(* IEC 61131-3 sources: lacyccom-procedural/src/drive_functions/blocks (part 4) *)

(* ---- LAcycCom_ReadDriveMessagesOperatingHours.st ---- *)
USING System.Timer;
USING System.DateTime;
USING System.Math;
USING Siemens.Simatic.Hardware.Utilities;
USING Siemens.Simatic.Clocks;

NAMESPACE Simatic.Ax.LAcycCom.Procedural
  TYPE
    LAcycCom_ReadDriveMessagesOperatingHoursStates : SINT (
      FB_IDLE := SINT#0,   // Idle state in FB
      FB_ALARMS_DATASET := SINT#1,   // Preparing dataset state in FB (alarms)
      FB_FAULTS_DATASET := SINT#2,   // Preparing dataset state in FB (faults)
      FB_ALARMS_GONE_DATASET := SINT#4,   // State that prepare dataset (r2125) and call ReadDriveParams
      FB_READ_STEP_1 := SINT#5,   // Call ReadDriveParams and write messages in statBuffer state
      FB_READ_STEP_2 := SINT#6,   // Call ReadDriveParams with FALSE state
      FB_SORTING := SINT#10   // Sorting state in FB
    ) := FB_IDLE;
  END_TYPE

  ///------------------------------------------------------------------------------
  /// SIEMENS AG
	/// (c)Copyright 2026 All Rights Reserved
	///-----------------------------------------------------------------------------
	/// Library: LAcycCom
	/// Tested with: S7-1513-1 PN
	/// Engineering: SIMATIC AX
	/// Restrictions: The drive must provide operating hours (days + ms)
	/// Requirements: S7-1200 / S7-1500
	///               FB LAcycCom_ResourceManager is required
	/// Functionality: Read alarms and faults from G120 drive (convert operating
	///                hours to "time" in reference to SIMATIC controller) and output
	///                in structure (newest elements first)
  ///------------------------------------------------------------------------------
  FUNCTION_BLOCK LAcycCom_ReadDriveMessagesOperatingHours
    {S7.Extern = ReadWrite}
    VAR_INPUT
      execute : BOOL;   /// TRUE: Rising edge starts the functionality once
      alarms : BOOL := TRUE;   /// TRUE: Enable reading of alarms
      faults : BOOL := TRUE;   /// TRUE: Enable reading of faults
      hardwareId : UINT;   /// Hardware identifier of the hardware module
    END_VAR

    {S7.Extern = ReadOnly}
    VAR_OUTPUT
      done : BOOL;   /// TRUE: Commanded action has been completed successfully
      busy : BOOL;   /// TRUE: FB is not finished and new output values can be expected
      error : BOOL;   /// TRUE: Rising edge informs that an error occurred during the execution of the FB
      status : LAcycCom_DriveFunctionStatus;   /// Status identifier
      diagnostics : LAcycCom_typeDriveDiagnostics;   /// Diagnostics structure
      messages : ARRAY[0..MESSAGES_COUNT_UPPER_LIM] OF LAcycCom_typeDriveMessage;   /// List of drive messages
    END_VAR

    VAR_IN_OUT
      requestBufferHeader : LAcycCom_typeRequestBufferHeader;   /// Interface for header of request buffer
      requestBuffer : ARRAY[*] OF LAcycCom_typeRequestBufferElement;   /// Interface for request buffer
    END_VAR

    VAR
      _busy : BOOL;   /// Static value for output busy
      _done : BOOL;   /// Static value for output done
      _error : BOOL;   /// Static value for output error
      _status : LAcycCom_DriveFunctionStatus;   /// Static value for output status
      _executeOld : BOOL;   /// Old value of execute for edge detection
      _fbstate : LAcycCom_ReadDriveMessagesOperatingHoursStates;   /// States in the function block state machine
      _alarmsInput : BOOL;   /// Static variable for input "alarms"
      _faultsInput : BOOL;   /// Static variable for input "faults"
      _driveObjectId : SINT;   /// Intern identification number of the drive object
      _hardwareId : UINT;   /// Intern hardware identifier of the hardware module
      _dtl : LDATE_AND_TIME;   /// Time varible for comparasion (sorting)
      _indexNew : DINT;   /// Index of newest elemet (for sorting)
      _offset : SINT;   /// Offset for statBuffer/ first empty element in statBuffer
      _warningNoMessages : BOOL;   /// TRUE: At least one of two inputs must be selected
      _warningRetriggering : BOOL;   /// TRUE: Input execute is set during processing
      _alarmsComplete : BOOL;   /// TRUE: FB_READ state complete successfully (alarms)
      _currentMessage : LAcycCom_DriveMessageType;   /// Static variable represents current message type
      _cpuTime : LDATE_AND_TIME;   /// Current data and current time-of-day of the CPU clock
      _cuTimeNotRead : BOOL;   /// TRUE: r2124 (represents system runtime total of CU ) is not yet read and evaluate
      _cpuTimeNotRead : BOOL;   /// TRUE: CPU time is not yet read
      _driveObjectTOD : TIME_OF_DAY;   /// Static variable represents r2124[0] - ms, convert to TOD
      _driveObjectDays : DINT;   /// Static variable represents r2124[1] - days
      _diffDays : DINT;   /// Difference in days between actual time from system runtime counter and time from come message
      _goneAlarms : ARRAY[0..ELEMENTS_COUNT_UPPER_LIM] OF BOOL;   /// TRUE: this alarm is already gone
      _dataset : ARRAY[0..PARAMETER_COUNT_READ_UPPER_LIM] OF LAcycCom_typeDriveDataset;   /// Dataset for LAcycCom_ReadDriveParams
      _buffer : ARRAY[0..MESSAGES_COUNT_UPPER_LIM] OF LAcycCom_typeDriveMessage;   /// Buffer for store alarms, faults and SI messages
      _instReadDriveParams : LAcycCom_ReadDriveParams;   /// Instance of LAcycCom_ReadDriveParams
    END_VAR

    VAR_TEMP
      tempIndex : DINT;   // Temporary loop index variable
      tempSort : SINT;   // Temporary loop variable for sorting
      tempUInt : UINT;   // Temporary UInt variable
      tempDriveObjectDays : DINT;   // Temporary variable for days
      tempDriveObjectTOD : TIME_OF_DAY;   // Temporary variable for data type TOD
      tempDays : DINT;
      tempTOD : TIME_OF_DAY;
      tempRetValWord : WORD;   // Return value of system function
      tempQuitient : DINT;   // Temporary variable for quititent
      tempRemainder : DINT;   // Temporary variable for remainder
      tempDTL : LDATE_AND_TIME;   // Temporary DTL variable
      tempGeoAddr : GeoAddr;   // Current Geo Address information
      tempVoidDiagnostics : LAcycCom_typeDriveDiagnostics;   // Temporary empty diagnostics structure
      tempVoidMessage : LAcycCom_typeDriveMessage; // Temporary empty message structure
    END_VAR

    VAR CONSTANT
      INT_ERR_NOT_CONFIG : WORD := WORD#16#8093;   // The DP component addressed via ID or F_ID is not configured (ReadRecord/WriteRecord)
      INT_ERR_NOT_KNOWN : WORD := WORD#16#80B0;   // Data record not known in module. Illegal data record number ≥ 256 (ReadRecord/WriteRecord)
      INT_ERR_LOG_START_ADDR : WORD := WORD#16#8090;   // Invalid logical start address (ReadRecord/WriteRecord)
      DO_NOT_EXIST : WORD := WORD#16#0019;   // Drive object does not exist
      OFFSET_INFO : SINT := SINT#8;   // Offset in dataset for "info" information
      OFFSET_DAYS : SINT := SINT#16;   // Offset in dataset for "Count days" information
      OFFSET_MS : SINT := SINT#24;   // Offset in dataset for "Count ms" information
      PARAMETER_COUNT_READ_UPPER_LIM : INT := INT#33;   // Count of parameters to be read in ReadDriveParams
      ELEMENTS_COUNT_UPPER_LIM : INT := INT#7;   // Count of elements in one message type
      INIT_DATASET : BYTE := BYTE#16#FF;   // Init value for dataset.errorValue
      MAX_COUNT_DAYS : DINT := DINT#24;   // Max count of days of data type "Time"
      DRIVE_OBJECT_ID_G120 : SINT := SINT#1;   // Drive object ID for G120 (e.g. CU240)
      MESSAGES_UPPER_LIM_LOCAL : INT := INT#15;   // Upper limit of elements in LAcycCom_typeDriveMessages
      DAYS_TO_MS : DINT := DINT#86400000;   // Constant to conversion from days to ms (1000*60*60*24)
      MESSAGES_COUNT_UPPER_LIM : INT := INT#23;   // Maxmimum number of messages
      TO_NS : LREAL := LREAL#1.0e+9 * 3600 * 24;   // Conversion value for days to ns
    END_VAR

    // Check if FB is triggered
    IF (execute = TRUE) AND (_executeOld = FALSE) AND (_busy = TRUE) THEN
      // Input execute is set during processing
      status := LAcycCom_DriveFunctionStatus#WARN_EXECUTE_SET_DURING_PROCESSING;
      _warningRetriggering := TRUE;
      _executeOld := execute;

    ELSIF (execute = TRUE) AND (_executeOld = FALSE) THEN
      // First call
      // Functionality is busy
      _busy := TRUE;

      // Reset other outputs
      _error := FALSE;
      _done := FALSE;
      _status := LAcycCom_DriveFunctionStatus#STATUS_FIRST_CALL;
      status := _status;

      busy := _busy;
      error := _error;
      done := _done;
      _executeOld := execute;

      // Initialize
      _alarmsInput := alarms;
      _faultsInput := faults;
      _driveObjectId := DRIVE_OBJECT_ID_G120;
      _hardwareId := hardwareId;
      _offset := SINT#0;
      _indexNew := SINT#0;
      diagnostics := tempVoidDiagnostics;
      diagnostics.firstParameterError := -1; // V1.3.2
      diagnostics.errorValue := BYTE#16#FF; // V1.3.2
      _warningNoMessages := FALSE;
      _warningRetriggering := FALSE;
      _currentMessage := LAcycCom_DriveMessageType#ALARM;
      _alarmsComplete := FALSE;
      // Set a default value to first entry in dataset
      _dataset[0].errorValue := INIT_DATASET;
      // Set init time for comparison (sorting)
      _dtl := tempDTL;
      _cpuTimeNotRead := TRUE;
      _cuTimeNotRead := TRUE;

        // Clearing static and output area for alarms, faults and SI messages
        FOR tempIndex := 0 TO MESSAGES_COUNT_UPPER_LIM DO
          _buffer[tempIndex] := tempVoidMessage;
        END_FOR;
      // Write diagnostics
      diagnostics.hardwareId := _hardwareId;
      diagnostics.driveObjectId := _driveObjectId;

      // Call ReadDriveParams with FALSE
      _instReadDriveParams(execute := FALSE,
                          requestBufferHeader := requestBufferHeader,
                          requestBuffer := requestBuffer,
                          dataset := _dataset);

      // Check if device hardware address exist
      tempRetValWord := ReadSlotFromHardwareID(hardwareId := _hardwareId,
                                          geoAddr := tempGeoAddr);

      // Check if everything is okay
      IF tempRetValWord <> WORD#16#0 THEN
        _error := TRUE;
        diagnostics.subfunctionStatus := tempRetValWord;
        _status := LAcycCom_DriveFunctionStatus#ERR_HW_ID;
        RETURN;

      END_IF;

      // Alarms or faults
      IF _faultsInput = TRUE THEN
        _fbstate := LAcycCom_ReadDriveMessagesOperatingHoursStates#FB_FAULTS_DATASET;
      ELSIF _alarmsInput = TRUE THEN
        _fbstate := LAcycCom_ReadDriveMessagesOperatingHoursStates#FB_ALARMS_GONE_DATASET;
      ELSE
        // Warning. At least one of two inputs must be selected
        _status := LAcycCom_DriveFunctionStatus#STATUS_FINISHED_NO_MSG_SELECTED;
        _fbstate := LAcycCom_ReadDriveMessagesOperatingHoursStates#FB_SORTING;
        _warningNoMessages := TRUE;
      END_IF;
      RETURN;

    // Check if FB is disabled (falling edge) after job is done or FB is in error state
    ELSIF (execute = FALSE AND _busy = FALSE) AND
      (_error = TRUE OR _done = TRUE)
    THEN
      // Error outputs are reset with falling edge of enable input
      _error := FALSE;

      // Enable and busy are reset with falling edge of enable input
      _done := FALSE;
      _busy := FALSE;

      // Write outputs
      _status := LAcycCom_DriveFunctionStatus#STATUS_NO_CALL;
      status := _status;
      busy := _busy;
      done := _done;
      error := _error;
      _fbstate := LAcycCom_ReadDriveMessagesOperatingHoursStates#FB_IDLE;

      _executeOld := execute;
      RETURN;

      // FB is currently executed and not finished
    ELSIF _busy = TRUE THEN
      _executeOld := execute;

      // FB is disabled
    ELSE
      _executeOld := execute;
      RETURN;
    END_IF;

    //----------------------------------------------------------------------------------------------
    IF (_busy = TRUE) AND (_error = FALSE) THEN  // Functionality running
      CASE _fbstate OF

        LAcycCom_ReadDriveMessagesOperatingHoursStates#FB_ALARMS_DATASET:
          // Preparing dataset for ReadDriveParams
          // Alarms
          FOR tempIndex := 0 TO ELEMENTS_COUNT_UPPER_LIM DO
            tempUInt := TO_UINT(tempIndex);
            // Index 0 ..7 - r2122 - "Alarm Code"
            _dataset[tempIndex].parameterNumber := UINT#2122;
            _dataset[tempIndex].index := tempUInt;
            // Index 8 ..15 - r2124 - "Alarm Info"
            _dataset[tempIndex + OFFSET_INFO].parameterNumber := UINT#2124;
            _dataset[tempIndex + OFFSET_INFO].index := tempUInt;
            // Index 16 .. 23 - r2145 - "Alarm come time in days"
            _dataset[tempIndex + OFFSET_DAYS].parameterNumber := UINT#2145;
            _dataset[tempIndex + OFFSET_DAYS].index := tempUInt;
            // Index 24 .. 31 - r2123 - "Alarm come time in ms"
            _dataset[tempIndex + OFFSET_MS].parameterNumber := UINT#2123;
            _dataset[tempIndex + OFFSET_MS].index := tempUInt;
          END_FOR;
          // r2114 - System Runtime Total. Index 32 and 33
          _dataset[32].parameterNumber := UINT#2114;
          _dataset[32].index := UINT#0;    // ms
          _dataset[33].parameterNumber := UINT#2114;
          _dataset[33].index := UINT#1;  // Days
          _fbstate := LAcycCom_ReadDriveMessagesOperatingHoursStates#FB_READ_STEP_1;
          _currentMessage := LAcycCom_DriveMessageType#ALARM;

        LAcycCom_ReadDriveMessagesOperatingHoursStates#FB_FAULTS_DATASET:
          // Preparing dataset for ReadDriveParams
          // Faults
          FOR tempIndex := 0 TO ELEMENTS_COUNT_UPPER_LIM DO
            tempUInt := TO_UINT(tempIndex);
            // Index 0 ..7 - r945 - "Fault Code"
            _dataset[tempIndex].parameterNumber := UINT#945;
            _dataset[tempIndex].index := tempUInt;
            // Index 8 ..15 - r949 - "Fault Info"
            _dataset[tempIndex + OFFSET_INFO].parameterNumber := UINT#949;
            _dataset[tempIndex + OFFSET_INFO].index := tempUInt;
            // Index 16 .. 23 - r2130 - "Fault come time in days"
            _dataset[tempIndex + OFFSET_DAYS].parameterNumber := UINT#2130;
            _dataset[tempIndex + OFFSET_DAYS].index := tempUInt;
            // Index 24 .. 31 - r948 - "Fault come time in ms"
            _dataset[tempIndex + OFFSET_MS].parameterNumber := UINT#948;
            _dataset[tempIndex + OFFSET_MS].index := tempUInt;
            _goneAlarms[tempIndex] := FALSE;
          END_FOR;

          // r2114 - System Runtime Total. Index 32 and 33
          _dataset[32].parameterNumber := UINT#2114;
          _dataset[32].index := UINT#0;    // ms
          _dataset[33].parameterNumber := UINT#2114;
          _dataset[33].index := UINT#1;  // Days
          _fbstate := LAcycCom_ReadDriveMessagesOperatingHoursStates#FB_READ_STEP_1;
          _currentMessage := LAcycCom_DriveMessageType#FAULT;

        LAcycCom_ReadDriveMessagesOperatingHoursStates#FB_ALARMS_GONE_DATASET:
          IF NOT _instReadDriveParams.busy AND
            NOT _instReadDriveParams.done AND
            NOT _instReadDriveParams.error
          THEN
            // Prepare dataset
            FOR tempIndex := 0 TO ELEMENTS_COUNT_UPPER_LIM DO
              tempUInt := TO_UINT(tempIndex);
              // Index 0..7 - r2125 - "Alarm time removed in milliseconds"
              _dataset[tempIndex].parameterNumber := UINT#2125;
              _dataset[tempIndex].index := tempUInt;
            END_FOR;

          END_IF;

          // Call ReadDriveParams
          _instReadDriveParams(execute := TRUE,
                              parameterCount := ELEMENTS_COUNT_UPPER_LIM + 1, //8 parameter
                              driveObjectId := _driveObjectId,
                              hardwareId := _hardwareId,
                              requestBufferHeader := requestBufferHeader,
                              requestBuffer := requestBuffer,
                              dataset := _dataset);

          IF NOT _instReadDriveParams.busy THEN
            diagnostics := _instReadDriveParams.diagnostics;
            IF _instReadDriveParams.done = TRUE THEN
              // To determine what alarms are already gone
              FOR tempIndex := 0 TO ELEMENTS_COUNT_UPPER_LIM DO
                IF _dataset[tempIndex].dwordValue <> WORD#16#0 THEN
                  _goneAlarms[tempIndex] := TRUE;
                ELSE
                  _goneAlarms[tempIndex] := FALSE; // 01.05.02
                END_IF;
              END_FOR;

              // Call ReadDriveParams with FALSE
              _instReadDriveParams(execute := FALSE,
                                  requestBufferHeader := requestBufferHeader,
                                  requestBuffer := requestBuffer,
                                  dataset := _dataset);
              // Go next
              _fbstate := LAcycCom_ReadDriveMessagesOperatingHoursStates#FB_ALARMS_DATASET;

            ELSIF _instReadDriveParams.error = TRUE THEN
              _error := TRUE;
              // HwId is wrong
              IF (_instReadDriveParams.status = LAcycCom_DriveFunctionStatus#ERR_WRITERECORD OR _instReadDriveParams.status = LAcycCom_DriveFunctionStatus#ERR_READRECORD) AND
                ((_instReadDriveParams.diagnostics.subfunctionStatus = INT_ERR_NOT_CONFIG)
                OR (_instReadDriveParams.diagnostics.subfunctionStatus = INT_ERR_NOT_KNOWN)
                OR (_instReadDriveParams.diagnostics.subfunctionStatus = INT_ERR_LOG_START_ADDR))
              THEN
                _status := LAcycCom_DriveFunctionStatus#ERR_HW_ID;
                // Drive object does not exist
              ELSIF _dataset[0].errorValue = DO_NOT_EXIST THEN
                _status := LAcycCom_DriveFunctionStatus#ERR_DO_ID;
              ELSE
                _status := LAcycCom_DriveFunctionStatus#ERR_READ_DRIVE_PARAMS_ALARMS_GONE;

              END_IF;

            END_IF;
          END_IF;

        LAcycCom_ReadDriveMessagesOperatingHoursStates#FB_READ_STEP_1:
          IF _cpuTimeNotRead = TRUE THEN
            // Read CPU time
            tempRetValWord := GetLocalDateTime(_cpuTime); // Reading current date and time of cpu clock

            // Error occurred during RD_LOC_T command
            IF (tempRetValWord <> WORD#16#0) AND (tempRetValWord <> WORD#16#0001) THEN
              _error := TRUE;
              diagnostics.subfunctionStatus := tempRetValWord;
              _status := LAcycCom_DriveFunctionStatus#ERR_GET_LOCAL_DATE_TIME;
            END_IF;
            _cpuTimeNotRead := FALSE;
          END_IF;

          // Call ReadDriveParams
          _instReadDriveParams(execute := TRUE,
                              parameterCount := PARAMETER_COUNT_READ_UPPER_LIM + 1, //34 parameter = 32 parameter for messages + 2 parameter for "System Runtime Total" r2124[0] and r2124[1]
                              driveObjectId := _driveObjectId,
                              hardwareId := _hardwareId,
                              requestBufferHeader := requestBufferHeader,
                              requestBuffer := requestBuffer,
                              dataset := _dataset);

          IF NOT _instReadDriveParams.busy THEN
            diagnostics := _instReadDriveParams.diagnostics;
            IF _instReadDriveParams.done = TRUE THEN
              // CU Time from parameter r2124
              IF _cuTimeNotRead = TRUE THEN
                _driveObjectDays := TO_DINT(_dataset[33].dwordValue);   // Days as DINT
                _driveObjectTOD := TO_TOD(TO_LWORD(TO_LINT(_dataset[32].dwordValue) * LINT#1000000)); // ms convert to TOD
                _cuTimeNotRead := FALSE;
              END_IF;
              // Copy to static area only elements with content
              FOR tempIndex := 0 TO ELEMENTS_COUNT_UPPER_LIM DO
                IF NOT _goneAlarms[tempIndex] THEN
                  _buffer[_offset].code := TO_UINT(_dataset[tempIndex].dwordValue);
                  // If parameter empty - then go next
                  IF _dataset[tempIndex].dwordValue = WORD#16#0 THEN
                    EXIT;
                  END_IF;

                  _buffer[_offset].info := TO_UDINT(_dataset[tempIndex + OFFSET_INFO].dwordValue);
                  tempDriveObjectDays := TO_DINT(_dataset[tempIndex + OFFSET_DAYS].dwordValue);
                  tempDriveObjectTOD := TO_TOD(TO_LWORD(_dataset[tempIndex + OFFSET_MS].dwordValue));
                  //=======================================================================================================================================
                  // Calcutation "come Date and Time" of G120. This CUs (all G120 except CU230P-2) have only system runtime counter...
                  // comeDateAndTime = CPU Time(statCPUTime) - (difference statCUDays and tempDays) - (difference statCUTOD and tempTOD)
                  _diffDays := _driveObjectDays - tempDriveObjectDays; // Difference in days between actual time from system runtime counter and time from come message
                  _buffer[_offset].comeDateAndTime := _cpuTime;
                  IF ABS(_diffDays) <= MAX_COUNT_DAYS THEN  // Max value of variable Time is T#24d
                    tempDays := (TO_DINT(TO_LWORD(_buffer[_offset].comeDateAndTime)) / DAYS_TO_MS) - _diffDays; // Difference drive object days to diff days
                    tempTOD := TO_TOD(_buffer[_offset].comeDateAndTime); // extract time of day from buffer
                    NewDateAndTime(TO_LDATE(TO_LWORD(tempDays)), TO_LTOD(tempTOD), _buffer[_offset].comeDateAndTime); // create new date and time based on day difference and current time of day

                  ELSE // When count of days > 24 then must be sliced
                    tempQuitient := _diffDays / MAX_COUNT_DAYS;
                    tempRemainder := _diffDays MOD MAX_COUNT_DAYS;
                    FOR tempSort := 1 TO TO_SINT(tempQuitient) DO
                      tempDays := (TO_DINT(TO_LWORD(_buffer[_offset].comeDateAndTime)) / DAYS_TO_MS) - (MAX_COUNT_DAYS * DAYS_TO_MS);
                      tempTOD := TO_TOD(_buffer[_offset].comeDateAndTime); // extract time of day from buffer
                      NewDateAndTime(TO_LDATE(TO_LWORD(tempDays)), TO_LTOD(tempTOD), _buffer[_offset].comeDateAndTime); // create new date and time based on day difference and current time of day
                    END_FOR;
                    tempDays := (TO_DINT(TO_LWORD(_buffer[_offset].comeDateAndTime)) / DAYS_TO_MS) - (tempRemainder * DAYS_TO_MS); // Difference statCUDays and tempDays in format Time
                    tempTOD := TO_TOD(_buffer[_offset].comeDateAndTime); // extract time of day from buffer
                    NewDateAndTime(TO_LDATE(TO_LWORD(tempDays)), TO_LTOD(tempTOD), _buffer[_offset].comeDateAndTime);
                  END_IF;

                  // tempTime := T_DIFF(IN1 := statDriveObjectTOD, IN2 := tempDriveObjectTOD); // Difference statCUTOD and tempTOD in format Time - ms
                  // statBuffer.comeDateAndTime[statOffset] := T_SUB(IN1 := statBuffer.comeDateAndTime[statOffset], IN2 := tempTime); // Subtraction ms

                  tempDays := TO_DINT(TO_LWORD(_driveObjectTOD)) - TO_DINT(TO_LWORD(tempDriveObjectTOD)) / DAYS_TO_MS; // Difference statCUTOD and tempTOD in format Time - ms
                  tempTOD := TO_TOD(_buffer[_offset].comeDateAndTime); // extract time of day from buffer
                  NewDateAndTime(TO_LDATE(TO_LWORD(tempDays)), TO_LTOD(tempTOD), _buffer[_offset].comeDateAndTime);

                  //=======================================================================================================================================
                  _buffer[_offset].messageType := _currentMessage; // Identifier for message
                  _offset := _offset + SINT#1;
                END_IF;
              END_FOR;
              // Set "complete" flag
              IF _currentMessage = LAcycCom_DriveMessageType#ALARM THEN
                _alarmsComplete := TRUE;
              END_IF;

              // Go next step
              _fbstate := LAcycCom_ReadDriveMessagesOperatingHoursStates#FB_READ_STEP_2;

              // Error while reading  with ReadDriveParams
            ELSIF _instReadDriveParams.error = TRUE THEN
              _error := TRUE;
              // HwId is wrong
              IF (_instReadDriveParams.status = LAcycCom_DriveFunctionStatus#ERR_WRITERECORD OR _instReadDriveParams.status = LAcycCom_DriveFunctionStatus#ERR_READRECORD) AND
                ((_instReadDriveParams.diagnostics.subfunctionStatus = INT_ERR_NOT_CONFIG)
                OR (_instReadDriveParams.diagnostics.subfunctionStatus = INT_ERR_NOT_KNOWN)
                OR (_instReadDriveParams.diagnostics.subfunctionStatus = INT_ERR_LOG_START_ADDR))
              THEN
                _status := LAcycCom_DriveFunctionStatus#ERR_HW_ID;
                // Drive object does not exist
              ELSIF _dataset[0].errorValue = DO_NOT_EXIST THEN
                _status := LAcycCom_DriveFunctionStatus#ERR_DO_ID;
              ELSE
                CASE _currentMessage OF
                  LAcycCom_DriveMessageType#ALARM:
                    _status := LAcycCom_DriveFunctionStatus#ERR_READ_DRIVE_PARAMS_ALARMS;
                  LAcycCom_DriveMessageType#FAULT:
                    _status := LAcycCom_DriveFunctionStatus#ERR_READ_DRIVE_PARAMS_FAULTS;
                  ELSE
                    ;
                END_CASE;
              END_IF;
            END_IF;
          END_IF;

          LAcycCom_ReadDriveMessagesOperatingHoursStates#FB_READ_STEP_2:
          // Call ReadDriveParams with FALSE
          _instReadDriveParams(execute := FALSE,
                              requestBufferHeader := requestBufferHeader,
                              requestBuffer := requestBuffer,
                              dataset := _dataset);

          // Choice next step. Right call order: faults, alarms
          IF (_alarmsInput AND NOT _alarmsComplete) THEN
            _fbstate := LAcycCom_ReadDriveMessagesOperatingHoursStates#FB_ALARMS_GONE_DATASET;
          ELSE
            _fbstate := LAcycCom_ReadDriveMessagesOperatingHoursStates#FB_SORTING;
          END_IF;

        LAcycCom_ReadDriveMessagesOperatingHoursStates#FB_SORTING:
          // When at least one message has been read
          IF _offset <> 0 THEN
            // Sorting algorithm. Newest message - first
            // When more then two messages of different type have the same come time, then order sequence is - alarms, faults, SI messages
            FOR tempSort := 0 TO (_offset - SINT#1) DO
              // Find newest element
              FOR tempIndex := 0 TO (_offset - 1) DO
                IF _buffer[tempIndex].comeDateAndTime >= _dtl THEN
                  _dtl := _buffer[tempIndex].comeDateAndTime;
                  _indexNew := tempIndex;
                END_IF;
              END_FOR;

              // Copy found element to output structure
              messages[tempSort] := _buffer[_indexNew];

              // Remove this element from buffer - by setting the value as small as possible
              _buffer[_indexNew].comeDateAndTime := tempDTL;
              // Set init time for next comparison
              _dtl := tempDTL;
            END_FOR;
          END_IF;
          // Set "done" flag
          _done := TRUE;

        ELSE
          _error := TRUE;
          _status := LAcycCom_DriveFunctionStatus#ERR_UNDEFINED_STATE;
      END_CASE;
    END_IF;

    //----------------------------------------------------------------------------------------------
    // Write outputs and error handling
    //----------------------------------------------------------------------------------------------
    // Error occurred in request
    IF _error = TRUE
    THEN
      _done := FALSE;
      _busy := FALSE;
      // Write diagnostics
      diagnostics.stateNumber := _fbstate;
      diagnostics.status := _status;

      // Request finished
    ELSIF _done = TRUE
    THEN
      _busy := FALSE;
      _error := FALSE;
      _fbstate := LAcycCom_ReadDriveMessagesOperatingHoursStates#FB_IDLE;
      // Set status
      IF _warningRetriggering = TRUE THEN
        // If input execute is set during processing
        _status := LAcycCom_DriveFunctionStatus#ERR_AMBIGUOUS_FB_CALL;
        diagnostics.status := _status;
        _error := TRUE;
        _done := FALSE;
      ELSIF _warningNoMessages = FALSE THEN
        // Execution finished without errors
        _status := LAcycCom_DriveFunctionStatus#STATUS_EXECUTION_FINISHED;
      ELSE
        // Warning. At least one of two inputs must be selected
        _status := LAcycCom_DriveFunctionStatus#STATUS_FINISHED_NO_MSG_SELECTED;
        diagnostics.status := _status;
      END_IF;

      // If input execute is set during processing
    ELSIF _warningRetriggering = TRUE
    THEN
      _status := LAcycCom_DriveFunctionStatus#WARN_EXECUTE_SET_DURING_PROCESSING;

      // Request in execution
    ELSE
      _status := LAcycCom_DriveFunctionStatus#STATUS_SUBSEQUENT_CALL;
    END_IF;

    // Write static values to outputs
    done := _done;
    busy := _busy;
    error := _error;
    status := _status;
  //----------------------------------------------------------------------------------------------
  END_FUNCTION_BLOCK
END_NAMESPACE

(* ---- LAcycCom_ReadDriveParams.st ---- *)
USING System.Timer;
USING Siemens.Simatic.DistributedIO;

NAMESPACE Simatic.Ax.LAcycCom.Procedural
  TYPE INTERNAL
    LAcycCom_ReadDriveParamsStates : SINT(
      FB_IDLE := SINT#0,   // Idle state in FB
      FB_FIRST_CYCLE := SINT#1,   // First cycle state in FB
      FB_ALLOCATE := SINT#2,   // Allocating a request element in request buffer DB
      FB_GET_RESOURCE := SINT#3,   // State to check if the communication to the drive object can be established
      FB_BUSY := SINT#4,   // Busy state in FB
      FB_RELEASE := SINT#5,   // State to return the allocated index
      FB_DONE := SINT#6,   // Done state in FB
      FB_ERROR := SINT#7,   // Error state in FB
      FB_BUSY_WriteRecord := SINT#8,   // WriteRecord in busy state
      FB_BUSY_ReadRecord := SINT#9,   // ReadRecord in busy state
      FB_BUSY_WAIT := SINT#10   // State when temporary error occurred
    ) := FB_IDLE;
  END_TYPE

  ///------------------------------------------------------------------------------------------
  /// SIEMENS AG
	/// (c)Copyright 2026 All Rights Reserved
	///------------------------------------------------------------------------------------------
	/// Library: LAcycCom
	/// Tested with: S7-1513-1 PN
	/// Engineering: SIMATIC AX
	/// Restrictions: ---
	/// Requirements: S7-1200 / S7-1500
	///               FB LAcycCom_ResourceManager is required
	/// Functionality: Reads parameters from a drive object according to the configured dataset
  ///------------------------------------------------------------------------------------------
  FUNCTION_BLOCK LAcycCom_ReadDriveParams
    {S7.extern = ReadWrite}
    VAR_INPUT
      execute : BOOL;   /// TRUE: Rising edge starts the functionality once
      parameterCount : INT := -1;   /// Count of parameters to read (-1: read all parameter in dataset)
      driveObjectId : INT := -1;   /// Optional: Identification number of the drive object (value <0: driveObjectId is not used, i.e. the corresponding drive object is only addressed via the hardwareId)
      hardwareId : UINT;   /// Hardware identifier of the hardware module
    END_VAR

    {S7.extern = ReadOnly}
    VAR_OUTPUT
      done : BOOL;   /// TRUE: Finished reading all parameters
      busy : BOOL;   /// TRUE: FB is not finished and new output values can be expected
      error : BOOL;   /// TRUE: Rising edge informs that an error occurred during the execution of the FB
      status : LAcycCom_DriveFunctionStatus;   /// Status identifier
      diagnostics : LAcycCom_typeDriveDiagnostics;   /// Diagnostics structure
    END_VAR

    VAR_IN_OUT
      requestBufferHeader : LAcycCom_typeRequestBufferHeader;   /// Interface for header of request buffer
      requestBuffer : ARRAY[*] OF LAcycCom_typeRequestBufferElement;   /// Interface for request buffer
      dataset : ARRAY[*] OF LAcycCom_typeDriveDataset;   /// Interface for dataset
    END_VAR

    VAR
      _executeOld : BOOL := FALSE;   /// TRUE: Indicates that the execute input in the previous cycle was set
      _busy : BOOL := FALSE;   /// Static value for output busy
      _done : BOOL := FALSE;   /// Static value for output done
      _error : BOOL := FALSE;   /// Static value for output error
      _cmdBusy : BOOL := FALSE;   /// TRUE: Process is not yet complete
      _cmdDone : BOOL := FALSE;   /// TRUE: Data record was transferred
      _cmdError : BOOL := FALSE;   /// TRUE: An error occurred during processing
      _timerStart : BOOL := FALSE;   /// TRUE: Starts OnDelay
      _hwId : UINT := UINT#0;   /// Intern hardware identifier of the hardware module
      _doId : BYTE := BYTE#16#00;   /// Intern identification number of the drive object
      _refNo : BYTE := BYTE#16#00;   /// Reference number of request
      _withoutResourceManager : BOOL := FALSE;   /// TRUE: No resource manager available; FALSE: Resource manager available
      _fbState : LAcycCom_ReadDriveParamsStates := LAcycCom_ReadDriveParamsStates#FB_IDLE;   /// States in the function block state machine
      _fbSubState : LAcycCom_ReadDriveParamsStates := LAcycCom_ReadDriveParamsStates#FB_BUSY_WriteRecord;   /// States in the function block during processing (busy state)
      _fbSubStateOld : LAcycCom_ReadDriveParamsStates := LAcycCom_ReadDriveParamsStates#FB_BUSY_WriteRecord;   /// Previous state when temporary error occurs
      _stateNumber : LAcycCom_ReadDriveParamsStates := LAcycCom_ReadDriveParamsStates#FB_IDLE;   /// State of the FB when error occurred
      _status : LAcycCom_DriveFunctionStatus := LAcycCom_DriveFunctionStatus#STATUS_NO_CALL;   /// Static value for output status
      _subfunctionStatus : WORD := WORD#16#0000;   /// Block status or error information
      _errorCount : UINT := UINT#0;   /// Error counter of retry request
      _allocatedIndex : INT := 0;   /// Allocated element index in the buffer DB
      _countOfElements : INT := 0;   /// Number of parameters in the dataset
      _firstParameterError : INT := -1;   /// Number of parameter at which the error occurred (-1: no parameter with error)
      _warningRetriggering : BOOL;   /// TRUE: Input execute is set during processing
      _dataRecordNo : DInt;   /// Used data record
      _lowerBoundDataSet : DINT;   /// Lower bound of dataset
      _upperBoundDataSet : DINT;   /// Upper bound of dataset
      _parameter : ARRAY[0..READ_PARAMETERS_UPPER_LIM] OF LAcycCom_typeParameter;
      _reqParameterInit : LAcycCom_typeParameterAddress := ( attribute := BYTE#16#10, elementNo := BYTE#16#01, parameterNo := UINT#0, index := UINT#0 );
      _reqParameterHeader : LAcycCom_typeParameterHeader;
      _reqParameterAddress : ARRAY[0..READ_PARAMETERS_UPPER_LIM] OF LAcycCom_typeParameterAddress;
      _respParameterHeader : LAcycCom_typeParameterHeader;
      _respParameterData : ARRAY[0..LENGTH_PARAMETER_TELEGRAM_UPPER_LIM] OF BYTE;
      _instWriteRecord : WriteRecord;   /// WriteRecord command
      _instReadRecord : ReadRecord;   /// ReadRecord command
      _instOnDelay : OnDelay;   /// OnDelay
    END_VAR

    VAR_TEMP
      tempExecute : BOOL;   // TRUE: Indicates that the execute input was set
      tempCmdValid : BOOL;   // TRUE: New data record was received and is valid
      tempStatusWord : WORD;   // Temporary status
      tempUDint : UDINT;   // Temporary udint variable
      tempWord : WORD;   // Temporary word variable
      tempParameterCount : INT;   // Temporary variable of the output parameterCount
      tempPointer : INT;   // Temporary pointer variable
      tempIndex : INT;   // Temporary loop index variable
      tempLastQueueElement : INT;   // Last element in queue
      tempCmdStatus : DWORD;   // Temporary status of WriteRecord and ReadRecord command
      tempDWord : DWORD;   // Temporary DWORD variable
      tempVoidDiagnostics : LAcycCom_typeDriveDiagnostics;   // Temporary empty diagnostics structure
      tempVoidHeader : LAcycCom_typeParameterHeader;   // Temporary empty header structure
      tempActualElement : LAcycCom_typeDriveDataset;   // Temporary element of the dataset
      tempRecord : ARRAY[0..239] OF BYTE;   // Temporary record buffer for WriteRecord and ReadRecord instruction
    END_VAR

    VAR CONSTANT
      NO_PARAMETER_ERROR : INT := -1;   // No parameter error in response telegram
      ALL_ELEMENTS_OCCUPIED : INT := -1;   // All buffer elements are occupied
      READ_PARAMETERS_UPPER_LIM : INT := 38;   // Maximum count of parameters
      LENGTH_PARAMETER_TELEGRAM_UPPER_LIM : INT := 233;   // Maximum length of telegram for parameter information in BYTE
      MAX_ERROR_COUNT : UINT := UINT#40;   // Maximum error counter
      TIMER_TEMP_ERROR : TIME := T#200MS;   // Waiting time until next system function block call
      TIMER_ALLOCATION : TIME := T#10S;   // Timer limit for allocating a request element
      MAX_DRIVE_OBJECT_NO : INT := 254;   // Maximum drive object number limited by SINAMICS p101
    END_VAR

    tempExecute := execute;

    //----------------------------------------------------------------------
    // Processing
    //----------------------------------------------------------------------
    // Rising edge of execute starts functionality
    IF (tempExecute = TRUE) AND (_executeOld = FALSE) AND (_busy = TRUE) THEN
      // Input execute is set during processing
      _status := LAcycCom_DriveFunctionStatus#WARN_EXECUTE_SET_DURING_PROCESSING;
      _warningRetriggering := TRUE;

    ELSIF (tempExecute = TRUE) AND (_executeOld = FALSE) THEN
      // First call
      // Initialisation
      _done := FALSE;
      _busy := TRUE;
      _error := FALSE;
      _countOfElements := 0;
      _allocatedIndex := 0;
      _hwId := UINT#0;
      _subfunctionStatus := WORD#16#0;
      _doId := BYTE#0;
      _dataRecordNo := 0;
      _stateNumber := LAcycCom_ReadDriveParamsStates#FB_IDLE;
      _firstParameterError := -1;
      _cmdBusy := FALSE;
      _cmdDone := FALSE;
      _cmdError := FALSE;
      _errorCount := UINT#0;
      _warningRetriggering := FALSE;
      _fbSubState := LAcycCom_ReadDriveParamsStates#FB_BUSY_WriteRecord;
      _fbState := LAcycCom_ReadDriveParamsStates#FB_FIRST_CYCLE;

      _instOnDelay(signal := FALSE,
             duration := TIMER_ALLOCATION);

      // Initialize boundaries of dataset
      _lowerBoundDataSet := LOWER_BOUND(dataset, 1);
      _upperBoundDataSet := UPPER_BOUND(dataset, 1);
      _countOfElements := TO_INT(GetCountOfElements(_lowerBoundDataSet, _upperBoundDataSet));

      // FB is currently inactive
    ELSIF (tempExecute = FALSE) AND (_busy = FALSE)
    THEN
      _error := FALSE;
      _busy := FALSE;
      _done := FALSE;
      _fbState := LAcycCom_ReadDriveParamsStates#FB_IDLE;

      IF ((_status = LAcycCom_DriveFunctionStatus#WARN_EXECUTE) AND (execute = FALSE)) OR (_status <> LAcycCom_DriveFunctionStatus#WARN_EXECUTE) THEN
        _status := LAcycCom_DriveFunctionStatus#STATUS_NO_CALL;
      END_IF;

    END_IF; // tempExecute AND statExecuteOld = FALSE

    //----------------------------------------------------------------------
    // State Machine
    //----------------------------------------------------------------------

    IF (_busy = TRUE) AND (_error = FALSE) THEN  // Functionality running
      CASE _fbState OF
        LAcycCom_ReadDriveParamsStates#FB_FIRST_CYCLE:  // First cycle state

          // Clearing the sending buffer
          _reqParameterHeader := tempVoidHeader;
          FOR tempIndex := 0 TO READ_PARAMETERS_UPPER_LIM DO
            _reqParameterAddress[tempIndex] := _reqParameterInit;
          END_FOR;

          // Clearing the receive buffer
         _respParameterHeader := tempVoidHeader;
          FOR tempIndex := 0 TO LENGTH_PARAMETER_TELEGRAM_UPPER_LIM DO
            _respParameterData[tempIndex] := BYTE#16#00;
          END_FOR;

          // Initialization after start
          IF driveObjectId < 0 THEN // V1.5
            _dataRecordNo := DINT#16#B02E; // Base Mode Parameter Access local; doId not relevant
            _doId := BYTE#0;

          ELSIF (driveObjectId <= MAX_DRIVE_OBJECT_NO)
            AND (driveObjectId <> 0)
          THEN // V1.5.2
            _dataRecordNo := 47; // Data record 47; Base Mode Parameter Access global
            _doId := TO_BYTE(driveObjectId);

          ELSE // V1.5.2
            // Wrong drive object ID at input
            _error := TRUE;
            _stateNumber := _fbState;
            _status := LAcycCom_DriveFunctionStatus#ERR_INVALID_DRIVE_OBJECT_ID;
            _fbState := LAcycCom_ReadDriveParamsStates#FB_ERROR;
          END_IF;

          _hwId := hardwareId;
          tempParameterCount := parameterCount;

          diagnostics := tempVoidDiagnostics;
          IF _status = LAcycCom_DriveFunctionStatus#WARN_EXECUTE THEN
            diagnostics.status := _status;
          END_IF;

          diagnostics.driveObjectId := TO_SINT(_doId);
          diagnostics.hardwareId := _hwId;
          diagnostics.firstParameterError := _firstParameterError; // V1.3.2
          diagnostics.errorValue := BYTE#16#FF; // V1.3.2

          // Reference number for next request
          _refNo := TO_BYTE(TO_UINT(_refNo) + UINT#1);

          IF _error THEN // V1.5.2: Check if error appeared
            ;

          // Next state is depending on the FB mode
          ELSIF (_withoutResourceManager = FALSE) THEN
            _status := LAcycCom_DriveFunctionStatus#STATUS_ALLOCATE;
            _fbState := LAcycCom_ReadDriveParamsStates#FB_ALLOCATE;

          ELSE
            _status := LAcycCom_DriveFunctionStatus#STATUS_BUSY;
            _fbState := LAcycCom_ReadDriveParamsStates#FB_BUSY;
            _fbSubState := LAcycCom_ReadDriveParamsStates#FB_BUSY_WriteRecord;
          END_IF;

          // Calculates the amount of parameters (only if no error occurs)
          IF (_error = FALSE) THEN
            // Calculates the count of elements in readDataset if numberOfParameters < 1
            IF (tempParameterCount < 1) AND
              (_countOfElements <= READ_PARAMETERS_UPPER_LIM)
            THEN
              diagnostics.parameterCount := _countOfElements;
            ELSIF (tempParameterCount >= 1) AND  // V1.3.2
              // Check if numberOfParameters <= 39
              (tempParameterCount <= READ_PARAMETERS_UPPER_LIM + 1) AND
              (_countOfElements >= tempParameterCount)
            THEN
              _countOfElements := tempParameterCount;
              diagnostics.parameterCount := _countOfElements;
            ELSE
              _error := TRUE;
              _stateNumber := _fbState;
              _status := LAcycCom_DriveFunctionStatus#ERR_NO_OF_PARAMETERS;
              _fbState := LAcycCom_ReadDriveParamsStates#FB_ERROR;
            END_IF;
          END_IF; // IF (statError = FALSE)

        LAcycCom_ReadDriveParamsStates#FB_ALLOCATE:
          // Allocation of a request element
          IF (requestBufferHeader.lockBuffer = FALSE) AND (requestBufferHeader.nextFreeElement >= requestBufferHeader.bufferLowerBound) AND (requestBufferHeader.nextFreeElement <= requestBufferHeader.bufferUpperBound) THEN
            requestBufferHeader.lockBuffer := TRUE;
            _allocatedIndex := requestBufferHeader.nextFreeElement;
            requestBuffer[_allocatedIndex].state := BYTE#16#00;
            requestBuffer[_allocatedIndex].state.%X0 := TRUE;
            requestBuffer[_allocatedIndex].hardwareId := _hwId;
            requestBuffer[_allocatedIndex].queueElementNext := -1;
            _timerStart := FALSE;
            _status := LAcycCom_DriveFunctionStatus#STATUS_GET_RESOURCE;
            _fbState := LAcycCom_ReadDriveParamsStates#FB_GET_RESOURCE;

            // Build up queue
            IF (requestBufferHeader.firstQueueElement >= 0) THEN
              // Find last queue element
              tempIndex := requestBufferHeader.firstQueueElement;
              WHILE (tempIndex >= 0) DO
                tempLastQueueElement := tempIndex;
                tempIndex := requestBuffer[tempIndex].queueElementNext;
              END_WHILE;

              // Insert into list after last element
              requestBuffer[tempLastQueueElement].queueElementNext := _allocatedIndex;
              requestBuffer[_allocatedIndex].queueElementPrevious := tempLastQueueElement;
            ELSE
              // Element is first element in queue
              requestBufferHeader.firstQueueElement := _allocatedIndex;
              requestBuffer[_allocatedIndex].queueElementPrevious := -1;
            END_IF;

            // Searching for the next free request element
            FOR tempIndex := requestBufferHeader.bufferLowerBound TO TO_INT(requestBufferHeader.bufferUpperBound) DO
              IF (requestBuffer[tempIndex].state.%X0 = FALSE) THEN
                requestBufferHeader.nextFreeElement := tempIndex;
                EXIT;
              END_IF;

              // All request elements are occupied
              IF (tempIndex = requestBufferHeader.bufferUpperBound) THEN
                requestBufferHeader.nextFreeElement := ALL_ELEMENTS_OCCUPIED;
              END_IF;
            END_FOR;

            requestBufferHeader.lockBuffer := FALSE;

          ELSIF (_instOnDelay.output = TRUE) THEN
            _error := TRUE;
            _stateNumber := _fbState;
            _status := LAcycCom_DriveFunctionStatus#ERR_ALLOCATION_TIME;
            _fbState := LAcycCom_ReadDriveParamsStates#FB_ERROR;

          ELSE
            ; // Waiting until lockbit is reset and a request element is available
          END_IF; // (buffer.lockBuffer = FALSE) AND (buffer.actualWriteIndex >= 0)

          _instOnDelay(signal := _timerStart,
                 duration := TIMER_ALLOCATION);

          _timerStart := TRUE;
          IF (_instOnDelay.output = TRUE) THEN
            _timerStart := FALSE;
          END_IF;

        LAcycCom_ReadDriveParamsStates#FB_GET_RESOURCE:

          // Check buffer index for correctness
          IF (_allocatedIndex < requestBufferHeader.bufferLowerBound) OR (_allocatedIndex > requestBufferheader.bufferUpperBound) THEN
            _error := TRUE;
            _stateNumber := _fbState;
            _status := LAcycCom_DriveFunctionStatus#ERR_INVALID_BUF_INDEX;
            _fbState := LAcycCom_ReadDriveParamsStates#FB_ERROR;

          ELSE
            IF (requestBuffer[_allocatedIndex].state.%X0 = FALSE) OR
              (requestBuffer[_allocatedIndex].state.%X3 = TRUE)
            THEN
              // Request was rejected by buffer manager
              _error := TRUE;
              _stateNumber := _fbState;
              _status := LAcycCom_DriveFunctionStatus#ERR_REQUEST_REJECTED;
              _fbState := LAcycCom_ReadDriveParamsStates#FB_ERROR;

            ELSIF (requestBuffer[_allocatedIndex].state.%X2 = TRUE) THEN
              // Request already released
              _error := TRUE;
              _stateNumber := _fbState;
              _status := LAcycCom_DriveFunctionStatus#ERR_RESOURCE_RELEASED;
              _fbState := LAcycCom_ReadDriveParamsStates#FB_ERROR;

            ELSIF (requestBuffer[_allocatedIndex].state.%X1 = TRUE) THEN
              // Element is enabled
              _status := LAcycCom_DriveFunctionStatus#STATUS_BUSY;
              _fbState := LAcycCom_ReadDriveParamsStates#FB_BUSY;
              _fbSubState := LAcycCom_ReadDriveParamsStates#FB_BUSY_WriteRecord;

            ELSE
              // Element not enabled yet
              //
              _status := LAcycCom_DriveFunctionStatus#STATUS_GET_RESOURCE;
            END_IF;

          END_IF;

        LAcycCom_ReadDriveParamsStates#FB_BUSY:

          IF ((requestBuffer[_allocatedIndex].state.%X1 = TRUE) AND (_withoutResourceManager = FALSE) AND
            (requestBuffer[_allocatedIndex].state.%X3 = FALSE)) OR (_withoutResourceManager = TRUE)
          THEN
            CASE _fbSubState OF
              LAcycCom_ReadDriveParamsStates#FB_BUSY_WriteRecord:  // Writing the dataset configuration into the drive object

                IF (_cmdBusy = FALSE) THEN
                  // Resets WriteRecord command
                  _instWriteRecord(request := FALSE,
                               record := tempRecord);

                  // Creating header data
                  _reqParameterHeader.refNo := _refNo; // Telegram reference number
                  _reqParameterHeader.reqId := BYTE#16#01;  // 0x01 = request parameters
                  _reqParameterHeader.doId := _doId;  // Drive object identification number
                  _reqParameterHeader.parameterNo := TO_BYTE(_countOfElements);  // Count of parameters

                  // Copying the dataset into a static variable
                  FOR tempIndex := 0 TO _countOfElements - 1 DO
                    // begin at lower bound of dataset
                    tempActualElement := dataset[tempIndex + _lowerBoundDataSet];

                    // write common parameters
                    _parameter[tempIndex].index := tempActualElement.index;
                    _parameter[tempIndex].parameterNo := tempActualElement.parameterNumber;
                    _reqParameterAddress[tempIndex].index := _parameter[tempIndex].index;  // Subindex of parameter
                    _reqParameterAddress[tempIndex].parameterNo := _parameter[tempIndex].parameterNo;  // Parameter number
                  END_FOR;
                END_IF; // statCmdBusy = FALSE

                SerializeParamAddress(header := _reqParameterHeader, address := _reqParameterAddress, buffer := tempRecord);

                // WriteRecord command
                _instWriteRecord(request := TRUE,             // Transfer data record
                             hardwareId := _hwId,      // ID number of the hardware component
                             index := _dataRecordNo,   // Data record number
                             length := UINT#0,            // Maximum length of the data record to be transferred in bytes
                             record := tempRecord,        // Data record
                             done => _cmdDone,         // Data record was transferred
                             busy => _cmdBusy,         // The writing process is not yet complete
                             error => _cmdError,       // An error occurred during the writing process
                             status => tempCmdStatus);    // Status[1] = Error => Status[2] Error Decode + Status[3] Error Code

                // Error occurred
                IF (_cmdError = TRUE) AND (_error = FALSE) THEN
                  tempStatusWord.%B0 := tempCmdStatus.%B1;
                  tempStatusWord.%B1 := tempCmdStatus.%B2;

                  //Temporary command status (80A1, 80A7, 80B5, 80C0, 80C1, 80C2, 80C3 oder 80C4) are valid and retry command
                  IF (tempStatusWord = WORD#16#80A1) OR  // Negative acknowledgment when writing to the module
                    (tempStatusWord = WORD#16#80A7) OR   // DP slave or module is occupied (temporary error)
                    (tempStatusWord = WORD#16#80B5) OR   // DP slave or module not ready
                    (tempStatusWord = WORD#16#80C0) OR   // The data can only be written when the CPU is in STOP mode. Note: this means that writing by the user program is not possible. You can only write the data online with PG/PC.
                    (tempStatusWord = WORD#16#80C1) OR   // The data of the previous write job on the module for the same data record have not yet been processed by the module.
                    (tempStatusWord = WORD#16#80C2) OR   // The module is currently processing the maximum possible number of jobs for a CPU.
                    (tempStatusWord = WORD#16#80C3) OR   // The required operating resources are currently occupied.
                    (tempStatusWord = WORD#16#80C4) THEN // Internal temporary error. Job could not be executed. Repeat the job. If this error occurs often, check your installation for sources of electrical interference.

                    IF (_errorCount >= MAX_ERROR_COUNT) THEN
                      _error := TRUE;
                      _stateNumber := _fbSubState;
                      _subfunctionStatus := tempStatusWord;
                      _status := LAcycCom_DriveFunctionStatus#ERR_WRITERECORD_TEMP_COUNTER;
                      _fbState := LAcycCom_ReadDriveParamsStates#FB_ERROR;
                    ELSE
                      _errorCount := _errorCount + UINT#1;  // Increment internal error counter
                      _fbSubStateOld := LAcycCom_ReadDriveParamsStates#FB_BUSY_WriteRecord;
                      _fbSubState := LAcycCom_ReadDriveParamsStates#FB_BUSY_WAIT;
                    END_IF;
                  ELSE
                    _error := TRUE;
                    _stateNumber := _fbSubState;
                    _subfunctionStatus := tempStatusWord;
                    _status := LAcycCom_DriveFunctionStatus#ERR_WRITERECORD;
                    _fbState := LAcycCom_ReadDriveParamsStates#FB_ERROR;
                  END_IF;

                ELSIF (_cmdDone = TRUE) AND (_error = FALSE) THEN  // Processing completed without errors
                  _errorCount := UINT#0;  // V1.5.1 Reset error counter
                  _fbSubState := LAcycCom_ReadDriveParamsStates#FB_BUSY_ReadRecord; // WriteRecord completed and continue with ReadRecord
                END_IF; // statCmdError = TRUE

              LAcycCom_ReadDriveParamsStates#FB_BUSY_ReadRecord:  // Reading the values from the drive object
                // Resets ReadRecord command
                IF (_cmdBusy = FALSE) THEN
                  _instReadRecord(request := FALSE,
                            record := tempRecord);
                END_IF;

                _instReadRecord(request := TRUE,            // Transfer data record
                            hardwareId := _hwId,     // ID number of the hardware component
                            index := _dataRecordNo,  // Data record number
                            maxLength := UINT#0,        // Maximum length in bytes of the data record information to be read
                            record := tempRecord,       // Destination area for the data record read
                            valid => tempCmdValid,      // New data record was received and is valid
                            busy => _cmdBusy,        // The reading process is not yet complete
                            error => _cmdError,      // An error occurred during the reading process
                            status => tempCmdStatus);   // Status[1] = Error => Status[2] Error Decode + Status[3] Error Code

                tempUDint := DeserializeParamResponse(header => _respParameterHeader, response => _respParameterData, buffer := tempRecord);

                IF tempUDint > UDINT#0 THEN
                  // Error occurred
                  IF (_cmdError = TRUE) THEN
                    // Get the error information from the status information
                    tempStatusWord.%B0 := tempCmdStatus.%B1;
                    tempStatusWord.%B1 := tempCmdStatus.%B2;

                    //Temporary command status (80A0, 80A7, 80B5, 80C0, 80C1, 80C2, 80C3 oder 80C4) are valid and retry command
                    IF (tempStatusWord = WORD#16#80A0) OR  // Negative acknowledgment when reading the module
                      (tempStatusWord = WORD#16#80A7) OR   // DP slave or module is occupied (temporary error)
                      (tempStatusWord = WORD#16#80B5) OR   // DP slave or module not ready
                      (tempStatusWord = WORD#16#80C0) OR   // The data can only be written when the CPU is in STOP mode. Note: this means that writing by the user program is not possible. You can only write the data online with PG/PC.
                      (tempStatusWord = WORD#16#80C1) OR   // The data of the previous write job on the module for the same data record have not yet been processed by the module.
                      (tempStatusWord = WORD#16#80C2) OR   // The module is currently processing the maximum possible number of jobs for a CPU.
                      (tempStatusWord = WORD#16#80C3) OR   // The required operating resources are currently occupied.
                      (tempStatusWord = WORD#16#80C4) THEN // Internal temporary error. Job could not be executed. Repeat the job. If this error occurs often, check your installation for sources of electrical interference.

                      IF (_errorCount >= MAX_ERROR_COUNT) THEN
                        _error := TRUE;
                        _stateNumber := _fbSubState;
                        _subfunctionStatus := tempStatusWord;
                        _status := LAcycCom_DriveFunctionStatus#ERR_READRECORD_TEMP_COUNTER;
                        _fbState := LAcycCom_ReadDriveParamsStates#FB_ERROR;
                      ELSE
                        _errorCount := _errorCount + UINT#1;  // Increment internal error counter
                        _fbSubStateOld := LAcycCom_ReadDriveParamsStates#FB_BUSY_ReadRecord;
                        // V1.3.2. If error 80A0 then should be retry with WriteRecord command
                        IF (tempStatusWord = WORD#16#80A0) THEN
                          _fbSubStateOld := LAcycCom_ReadDriveParamsStates#FB_BUSY_WriteRecord;
                        END_IF;
                        _fbSubState := LAcycCom_ReadDriveParamsStates#FB_BUSY_WAIT;
                      END_IF; // statErrorCount >= MAX_ERROR_COUNT
                    ELSE
                      _error := TRUE;
                      _stateNumber := _fbSubState;
                      _subfunctionStatus := tempStatusWord;
                      _status := LAcycCom_DriveFunctionStatus#ERR_READRECORD;
                      _fbState := LAcycCom_ReadDriveParamsStates#FB_ERROR;
                    END_IF;

                    // Error : Reference number of the request does not match with the response reference number
                  ELSIF (_cmdBusy = FALSE) AND
                    (_refNo <> _respParameterHeader.refNo) AND
                    (tempCmdValid = TRUE) THEN

                    _error := TRUE;
                    _stateNumber := _fbSubState;
                    _status := LAcycCom_DriveFunctionStatus#ERR_REFERENCE_NO;
                    _fbState := LAcycCom_ReadDriveParamsStates#FB_ERROR;

                    // Error : Invalid response from the drive object (reqId: 16#01 - reading parameter successful; 16#81: reading parameter finished with error)
                  ELSIF NOT (_respParameterHeader.reqId = BYTE#16#81 OR _respParameterHeader.reqId = BYTE#16#01) AND
                    (_cmdBusy = FALSE) AND
                    (tempCmdValid = TRUE) THEN
                    _error := TRUE;
                    _stateNumber := _fbSubState;
                    _status := LAcycCom_DriveFunctionStatus#ERR_RESPONSE_ID;
                    _fbState := LAcycCom_ReadDriveParamsStates#FB_ERROR;

                    // Error : The received number of parameters does not match with the requested number of parameters
                  ELSIF (_cmdBusy = FALSE) AND
                    (_countOfElements <> TO_INT(_respParameterHeader.parameterNo)) AND
                    (tempCmdValid = TRUE) THEN

                    _error := TRUE;
                    _stateNumber := _fbSubState;
                    _status := LAcycCom_DriveFunctionStatus#ERR_PARAMETER_NO;
                    _fbState := LAcycCom_ReadDriveParamsStates#FB_ERROR;

                    // Error : The drive object does not match with the responsed DO
                  ELSIF (_cmdBusy = FALSE) AND
                    (_doId <>_respParameterHeader.doId) AND
                    (tempCmdValid = TRUE) THEN

                    _error := TRUE;
                    _stateNumber := _fbSubState;
                    _status := LAcycCom_DriveFunctionStatus#ERR_DRIVE_OBJECT_NO;
                    _fbState := LAcycCom_ReadDriveParamsStates#FB_ERROR;

                    // No error occurred during reading parameters
                  ELSIF (tempCmdValid = TRUE) THEN
                    // Analyse of the response buffer
                    tempPointer := 0;
                    FOR tempIndex := 0 TO _countOfElements - 1 DO
                      _parameter[tempIndex].format := _respParameterData[tempPointer];  // Format of the parameter

                      // Format = Error
                      IF (((TO_SINT(_respParameterData[tempPointer]) > LAcycCom_DriveValueFormats#FORMAT_DOUBLE_WORD) OR
                        ((TO_SINT(_respParameterData[tempPointer]) > LAcycCom_DriveValueFormats#FORMAT_FLOATING_POINT) AND (TO_SINT(_respParameterData[tempPointer]) < LAcycCom_DriveValueFormats#FORMAT_OCTET_STRING)) OR
                        ((TO_SINT(_respParameterData[tempPointer]) > LAcycCom_DriveValueFormats#FORMAT_OCTET_STRING) AND (TO_SINT(_respParameterData[tempPointer]) < LAcycCom_DriveValueFormats#FORMAT_TIME_DIFFERENCE)) OR
                        // V1.5.4 ((TO_SINT(_respParameterData[tempPointer]) > LAcycCom_DriveValueFormats#FORMAT_TIME_DIFFERENCE) AND (TO_SINT(_respParameterData[tempPointer]) < LAcycCom_DriveValueFormats#FORMAT_BYTE)) OR
                        ((TO_SINT(_respParameterData[tempPointer]) > LAcycCom_DriveValueFormats#FORMAT_TIME_DIFFERENCE) AND (TO_SINT(_respParameterData[tempPointer]) < LAcycCom_DriveValueFormats#FORMAT_TIME_DIFFERENCE_WO_DATE)) OR // V1.5.4: format "TimeDifference without date indication" added
                        ((TO_SINT(_respParameterData[tempPointer]) > LAcycCom_DriveValueFormats#FORMAT_TIME_DIFFERENCE_WO_DATE) AND (TO_SINT(_respParameterData[tempPointer]) < LAcycCom_DriveValueFormats#FORMAT_BYTE)) OR // V1.5.4: format "TimeDifference without date indication" added
                        (TO_SINT(_respParameterData[tempPointer]) < LAcycCom_DriveValueFormats#FORMAT_INTEGER_8))) AND (TO_SINT(_respParameterData[tempPointer]) <> LAcycCom_DriveValueFormats#FORMAT_ZERO)
                      THEN

                        // Format = Error, summarize the first and second error byte in a word error variable for each parameter
                        _parameter[tempIndex].errorValue := _respParameterData[tempPointer + 3];
                        IF (_firstParameterError = NO_PARAMETER_ERROR) THEN
                          diagnostics.firstParameterError := tempIndex;
                          diagnostics.errorValue := _parameter[tempIndex].errorValue; // V1.3.2
                          _firstParameterError := tempIndex;
                          _error := TRUE;
                          _stateNumber := _fbSubState;
                          _status := LAcycCom_DriveFunctionStatus#ERR_PARAMETER;
                          _fbState := LAcycCom_ReadDriveParamsStates#FB_ERROR;
                        END_IF;
                        // Points to the next parameter address
                        tempPointer := tempPointer + 6;
                      ELSE
                        CASE TO_SINT(_respParameterData[tempPointer]) OF
                          LAcycCom_DriveValueFormats#FORMAT_INTEGER_8:
                            _parameter[tempIndex].realValue := TO_REAL(TO_SINT(_respParameterData[tempPointer + 2]));
                            _parameter[tempIndex].dwordValue := _respParameterData[tempPointer + 2];
                            _parameter[tempIndex].errorValue := BYTE#16#FF; // Sets the error status and diagnostics

                            tempPointer := tempPointer + 4; // Points to the next parameter address

                          LAcycCom_DriveValueFormats#FORMAT_INTEGER_16:
                            tempWord.%B0 := _respParameterData[tempPointer + 3];
                            tempWord.%B1 := _respParameterData[tempPointer + 2];

                            _parameter[tempIndex].realValue := TO_REAL(TO_INT(tempWord));
                            _parameter[tempIndex].dwordValue := tempWord;
                            _parameter[tempIndex].errorValue := BYTE#16#FF; // Sets the error status and diagnostics

                            tempPointer := tempPointer + 4; // Points to the next parameter address

                          LAcycCom_DriveValueFormats#FORMAT_INTEGER_32:
                            tempDWord.%B0 := _respParameterData[tempPointer + 5];
                            tempDWord.%B1 := _respParameterData[tempPointer + 4];
                            tempDWord.%B2 := _respParameterData[tempPointer + 3];
                            tempDWord.%B3 := _respParameterData[tempPointer + 2];

                            _parameter[tempIndex].realValue := TO_REAL(tempDWord);
                            _parameter[tempIndex].dwordValue := tempDWord;
                            _parameter[tempIndex].errorValue := BYTE#16#FF; // Sets the error status and diagnostics

                            tempPointer := tempPointer + 6; // Points to the next parameter address

                          LAcycCom_DriveValueFormats#FORMAT_UNSIGNED_8, LAcycCom_DriveValueFormats#FORMAT_OCTET_STRING: // V1.5 change OCTET_STRING
                            _parameter[tempIndex].realValue := TO_REAL(TO_SINT(_respParameterData[tempPointer + 2]));
                            _parameter[tempIndex].dwordValue := _respParameterData[tempPointer + 2];
                            _parameter[tempIndex].errorValue := BYTE#16#FF; // Sets the error status and diagnostics

                            tempPointer := tempPointer + 4; // Points to the next parameter address

                          LAcycCom_DriveValueFormats#FORMAT_UNSIGNED_16:
                            tempWord.%B0 := _respParameterData[tempPointer + 3];
                            tempWord.%B1 := _respParameterData[tempPointer + 2];

                            _parameter[tempIndex].realValue := TO_REAL(TO_INT(tempWord));
                            _parameter[tempIndex].dwordValue := tempWord;
                            _parameter[tempIndex].errorValue := BYTE#16#FF; // Sets the error status and diagnostics

                            tempPointer := tempPointer + 4; // Points to the next parameter address

                          LAcycCom_DriveValueFormats#FORMAT_UNSIGNED_32, LAcycCom_DriveValueFormats#FORMAT_TIME_DIFFERENCE, LAcycCom_DriveValueFormats#FORMAT_TIME_DIFFERENCE_WO_DATE: // V1.5.4: format "TimeDifference without date indication" added
                            tempDWord.%B0 := _respParameterData[tempPointer + 5];
                            tempDWord.%B1 := _respParameterData[tempPointer + 4];
                            tempDWord.%B2 := _respParameterData[tempPointer + 3];
                            tempDWord.%B3 := _respParameterData[tempPointer + 2];

                            _parameter[tempIndex].realValue := TO_REAL(tempDWord);
                            _parameter[tempIndex].dwordValue := tempDWord;
                            _parameter[tempIndex].errorValue := BYTE#16#FF; // Sets the error status and diagnostics

                            tempPointer := tempPointer + 6; // Points to the next parameter address

                          LAcycCom_DriveValueFormats#FORMAT_FLOATING_POINT, LAcycCom_DriveValueFormats#FORMAT_DOUBLE_WORD:
                            tempDWord.%B0 := _respParameterData[tempPointer + 5];
                            tempDWord.%B1 := _respParameterData[tempPointer + 4];
                            tempDWord.%B2 := _respParameterData[tempPointer + 3];
                            tempDWord.%B3 := _respParameterData[tempPointer + 2];

                            _parameter[tempIndex].realValue := TO_REAL(tempDWord);
                            _parameter[tempIndex].dwordValue := tempDWord;
                            _parameter[tempIndex].errorValue := BYTE#16#FF; // Sets the error status and diagnostics

                            tempPointer := tempPointer + 6; // Points to the next parameter address

                          LAcycCom_DriveValueFormats#FORMAT_BYTE:
                            _parameter[tempIndex].realValue := TO_REAL(TO_DWORD(_respParameterData[tempPointer + 2]));
                            _parameter[tempIndex].dwordValue := _respParameterData[tempPointer + 2];
                            _parameter[tempIndex].errorValue := BYTE#16#FF; // Sets the error status and diagnostics

                            tempPointer := tempPointer + 4; // Points to the next parameter address

                          LAcycCom_DriveValueFormats#FORMAT_WORD:
                            tempWord.%B0 := _respParameterData[tempPointer + 3];
                            tempWord.%B1 := _respParameterData[tempPointer + 2];

                            _parameter[tempIndex].realValue := TO_REAL(TO_INT(tempWord));
                            _parameter[tempIndex].dwordValue := tempWord;
                            _parameter[tempIndex].errorValue := BYTE#16#FF; // Sets the error status and diagnostics

                            tempPointer := tempPointer + 4; // Points to the next parameter address

                          ELSE
                            ;
                        END_CASE;

                      END_IF; // Format = Error
                    END_FOR; // Analyse of the response buffer

                    // Copying parameter data into the dataset
                    FOR tempIndex := 0 TO _countOfElements - 1 DO
                      // begin at lower bound of dataset
                      tempActualElement := dataset[tempIndex + _lowerBoundDataSet];

                      // copy response into element
                      tempActualElement.index := _parameter[tempIndex].index;
                      tempActualElement.parameterNumber := _parameter[tempIndex].parameterNo;
                      tempActualElement.dwordValue := _parameter[tempIndex].dwordValue;
                      tempActualElement.realValue := _parameter[tempIndex].realValue;
                      tempActualElement.errorValue := _parameter[tempIndex].errorValue;

                      // copy element back to dataset
                      dataset[tempIndex + _lowerBoundDataSet] := tempActualElement;
                    END_FOR;

                    _cmdBusy := FALSE;
                    _cmdError := FALSE;

                    // Next state is depending on the FB mode
                    IF (_withoutResourceManager = FALSE) AND (_error = FALSE) THEN
                      _status := LAcycCom_DriveFunctionStatus#STATUS_RELEASE;
                      _fbState := LAcycCom_ReadDriveParamsStates#FB_RELEASE;

                    ELSIF (_error = FALSE) THEN
                      _status := LAcycCom_DriveFunctionStatus#STATUS_EXECUTION_FINISHED;
                      _fbState := LAcycCom_ReadDriveParamsStates#FB_DONE;

                    END_IF; // statMode = MODE_WITH_BUFFER_MANAGER
                  END_IF; // statCmdError = TRUE
                ELSE
                  _error := TRUE;
                  _stateNumber := _fbSubState;
                  _status := LAcycCom_DriveFunctionStatus#ERR_MISSMATCH_READ_BUFFER_SIZE;
                  _fbState := LAcycCom_typeDriveActDeactStates#FB_ERROR;
                END_IF;

              LAcycCom_ReadDriveParamsStates#FB_BUSY_WAIT:
                // Timer for temporary errors
                _instOnDelay(signal := _timerStart,
                             duration := TIMER_TEMP_ERROR);

                _timerStart := TRUE;
                IF (_instOnDelay.output = TRUE) THEN
                  _timerStart := FALSE;
                  _fbSubState := _fbSubStateOld;
                END_IF;

              ELSE
                _error := TRUE;
                _status := LAcycCom_DriveFunctionStatus#ERR_UNDEFINED_SUBSTATE;
                _stateNumber := _fbState;
                _fbState := LAcycCom_ReadDriveParamsStates#FB_ERROR;
            END_CASE;

          ELSE
            _error := TRUE;
            _status := LAcycCom_DriveFunctionStatus#ERR_COMMAND_TIMEOUT;
            _stateNumber := _fbState;
            _fbState := LAcycCom_ReadDriveParamsStates#FB_ERROR;
          END_IF; // ((buffer.element[statAllocatedIndex].enable = TRUE) AND (statMode = MODE_WITH_BUFFER_MANAGER)) OR statMode = MODE_WITHOUT_BUFFER_MANAGER

        LAcycCom_ReadDriveParamsStates#FB_RELEASE:
          // Check buffer index for correctness
          IF (_allocatedIndex < requestBufferHeader.bufferLowerBound) OR (_allocatedIndex > requestBufferHeader.bufferUpperBound) THEN
            _error := TRUE;
            _status := LAcycCom_DriveFunctionStatus#ERR_INVALID_BUF_INDEX;
            _stateNumber := _fbState;
            _fbState := LAcycCom_ReadDriveParamsStates#FB_ERROR;

          ELSIF (requestBufferHeader.lockBuffer = FALSE) THEN // V1.5.1
            requestBufferHeader.lockBuffer := TRUE;
            IF (requestBuffer[_allocatedIndex].state.%X0 = TRUE) THEN
              requestBuffer[_allocatedIndex].state.%X2 := TRUE;
            ELSE
              ;
            END_IF;
            requestBufferHeader.lockBuffer := FALSE;
            _status := LAcycCom_DriveFunctionStatus#STATUS_EXECUTION_FINISHED;
            _fbState := LAcycCom_ReadDriveParamsStates#FB_DONE;

          END_IF;

        ELSE
          _error := TRUE;
          _status := LAcycCom_DriveFunctionStatus#ERR_UNDEFINED_STATE;
          _stateNumber := _fbState;
          _fbState := LAcycCom_ReadDriveParamsStates#FB_ERROR;
      END_CASE;

      // If input execute is set during processing
      IF _warningRetriggering = TRUE AND _error = FALSE THEN
        _status := LAcycCom_DriveFunctionStatus#WARN_EXECUTE_SET_DURING_PROCESSING;
      END_IF;

    END_IF;

    //----------------------------------------------------------------------
    // Error handling and write outputs
    //----------------------------------------------------------------------

    // Edge detection
    _executeOld := tempExecute;

    IF (_fbState = LAcycCom_ReadDriveParamsStates#FB_ERROR) THEN
      // Release the allocated element when error occurs
      IF (_stateNumber <> LAcycCom_ReadDriveParamsStates#FB_FIRST_CYCLE) AND (_stateNumber <> LAcycCom_ReadDriveParamsStates#FB_ALLOCATE)
        AND (_busy = TRUE) AND (_withoutResourceManager = FALSE)
      THEN
        IF requestBufferHeader.lockBuffer = FALSE THEN // V1.5.1
          requestBufferHeader.lockBuffer := TRUE;
          IF (requestBuffer[_allocatedIndex].state.%X0 = TRUE) THEN
            requestBuffer[_allocatedIndex].state.%X2 := TRUE;
          ELSE
            ;
          END_IF;
          requestBufferHeader.lockBuffer := FALSE;

          // Write diagnostics
          diagnostics.stateNumber := _stateNumber;
          diagnostics.subfunctionStatus := _subfunctionStatus;
          diagnostics.status := _status;
          _busy := FALSE;
          _done := FALSE;

        END_IF;

      ELSE
        // Write diagnostics
        diagnostics.stateNumber := _stateNumber;
        diagnostics.subfunctionStatus := _subfunctionStatus;
        diagnostics.status := _status;
        _busy := FALSE;
        _done := FALSE;
      END_IF;

      // FB finished request
    ELSIF (_fbState = LAcycCom_ReadDriveParamsStates#FB_DONE) THEN

      // Output for one cycle minimum
      IF (tempExecute = FALSE) AND (_done = TRUE) THEN
        _done := FALSE;
        _status := LAcycCom_DriveFunctionStatus#STATUS_NO_CALL;
        _fbState := LAcycCom_ReadDriveParamsStates#FB_IDLE;
      ELSE
        _done := TRUE;
        _busy := FALSE;
      END_IF;
      // If input execute is set during processing
      IF _warningRetriggering = TRUE THEN
        _status := LAcycCom_DriveFunctionStatus#ERR_AMBIGUOUS_FB_CALL;
        diagnostics.status := _status;
        _error := TRUE;
        _done := FALSE;
      END_IF;
    END_IF;

    IF _busy = FALSE OR _error = FALSE
    THEN  // V1.5.1
      error := _error;
      status := _status;
    END_IF;

    busy := _busy;
    done := _done;
  END_FUNCTION_BLOCK
END_NAMESPACE
